# EPICS autosave request: apps/scalerApp/Db/joergerN_settings.req
# FILE... joerger_scaler_settings.req
# USAGE.. CLAS12 Joerger Scaler fields autosave'd.
#
file scaler16m_settings.req         P=$(P),S=$(S)
file scaler16m_addons_settings.req  P=$(P),S=$(S)
